// TIA Portal V16 export
// export: Created 2021-05-17T13:48:16.4866854Z, ExportSetting WithDefaults, DisplayName Totally Integrated Automation Portal, DisplayVersion V16 Update 3, DisplayName TIA Portal Version Control Interface, DisplayVersion V16 Update 2, DisplayName TIA Portal Openness, DisplayVersion V16 Update 3, DisplayName STEP 7 Professional, DisplayVersion V16 Update 3, DisplayName STEP 7 Safety, DisplayVersion V16, DisplayName WinCC Professional, DisplayVersion V16 Update 3
VAR_GLOBAL   // PLC tag table "PAL_TestFC18001"
   FIC101_RAW AT %MW100 : Int;   // FIC101 - Instrument Simulation - RAW SIGNAL
   OVER_RANGE AT %M102.0 : Bool;
   UNDER_RANGE AT %M102.1 : Bool;
   OUT_OF_RANGE AT %M102.2 : Bool;
   SCALE_VALUE AT %MD110 : Real;
END_VAR
